TYPE "MatCountPar"
VERSION : 0.1
// Block: MatCountPar
   STRUCT
      FAK : LReal;
   END_STRUCT;

END_TYPE
